{attribute 'linkalways'} 
{attribute 'no_explicit_call' := 'This FB is a CLASS and must be accessed using methods or properties'}
{attribute 'enable_dynamic_creation'}
FUNCTION_BLOCK Node_F_VN_AddToContainerElements_TcVnRectangle_DINT EXTENDS VisionNode
VAR
    stValue : _TcVnRectangle_DINT;
    ipContainer : _ITcVnContainer;
    hrPrev : _HRESULT(S_OK);
    hresult : _HRESULT(S_OK);
END_VAR

METHOD PUBLIC  Clone : I_Node
VAR
    pNode : POINTER TO Node_F_VN_AddToContainerElements_TcVnRectangle_DINT;
END_VAR
pNode := __NEW(Node_F_VN_AddToContainerElements_TcVnRectangle_DINT);
Clone := pNode^;
END_METHOD

METHOD FB_init : BOOL
VAR_INPUT
    bInitRetains : BOOL; // if TRUE, the retain variables are initialized (warm start / cold start)
    bInCopyCode : BOOL;  // if TRUE, the instance afterwards gets moved into the copy code (online change)
END_VAR
AddInput('stValue', stValue);
AddInput('ipContainer', ipContainer);
AddInput('hrPrev', hrPrev);
AddOutput('ipContainer', ipContainer);
AddOutput('hresult',hresult);
END_METHOD

METHOD PROTECTED OnExecute
hresult.Value := F_VN_AddToContainerElements_TcVnRectangle_DINT(
    stValue := stValue.Value,
    ipContainer := ipContainer.Value,
    hrPrev:= hrPrev.Value);
END_METHOD

METHOD PUBLIC PreExecutionCheck
VAR_INPUT
    Check : I_PreExecutionChecks;
END_VAR
Check.IsTrue(ipContainer.IsValid, 'ipContainer must be a valid container');
Check.IsTrue(ipContainer.IsType(TC_GLOBAL_CONST_LIST.ContainerType_Vector_TcVnRectangle_DINT), 'ipContainer contains incorrect type');
END_METHOD

END_FUNCTION_BLOCK

(* stored: Version 1.1.0.1, ProductVersion 3.1.4026.13
   POU Node_F_VN_AddToContainerElements_TcVnRectangle_DINT: Id {091a72ab-599a-45eb-b13b-22135ad34b8e}, SpecialFunc None
   Folder Constructor: Id {b826ee09-5178-46fe-bc1d-8871bdec4aaa}
   Method Clone: Id {6650fc41-e505-4290-80dd-9586256de0cf}
   Method FB_init: Id {df5d656c-92f4-4715-8383-1987d1998b1e}
   Method OnExecute: Id {61349d5d-4863-4c67-86d3-1ab83ab51011}
   Method PreExecutionCheck: Id {620556ca-68e6-4553-b159-7f7bf29cb602} *)
